// Implicitly generated code : DO NOT EDIT
FUNCTION CheckBounds : DINT
VAR_INPUT
	index, lower, upper: DINT;
END_VAR

// Implicitly generated code : Only an Implementation suggestion
{noflow}
IF  index < lower THEN
	GVL.udiLowerCnt := GVL.udiLowerCnt + 1;
	IF GVL.udiLowerCnt >= 1000000 THEN
		GVL.udiLowerCnt := 0;
	END_IF
	CheckBounds := lower;
ELSIF  index > upper THEN
	GVL.udiUpperCnt := GVL.udiUpperCnt + 1;
	IF GVL.udiUpperCnt >= 1000000 THEN
		GVL.udiUpperCnt := 0;
	END_IF
	CheckBounds := upper;
ELSE  
	CheckBounds := index;
END_IF
{flow}

END_FUNCTION

(* stored: Version 1.1.0.1, ProductVersion 3.1.4024.11
   POU CheckBounds: Id {cc3b0a0e-e50d-4f16-af24-bcd8ec6b74bb}, SpecialFunc CheckBounds *)
